{attribute 'qualified_only'}
{attribute 'strict'}
{attribute 'to_string'}
TYPE E_StateSystem :
(
	NoReference		, 	// system has not been initialized
	Initialize		, 	// System is initializing
	LoadParameters	, 	// System is loading parameters from/to file
	Safe			, 	// System is in safety state
	Enable			, 	// System is enabling 
	Home			, 	// system is hominig 
	Resetting		, 	// System is resetting
	Idle			, 	// system is waiting for commands
	Manual			, 	// System is in manual mode
	SemiAuto		, 	// System is in semi auto mode
	Automatic		, 	// system is in automatic mode 
	Fault			,	// System is in Fault state
	PowerOff		// system is powering off
)INT;
END_TYPE

(* stored: Version 1.1.0.1, ProductVersion 3.1.4024.10
   EnumerationTextList E_StateSystem: Id {e1b3949c-1926-4ece-ac62-019c23745b70} *)
